PROGRAM STATE_MACHINE
VAR
	timer: TON;
END_VAR

IF ( CTRL.sdo = TRUE)THEN
	timer(IN:=TRUE);
	IF (timer.Q = TRUE) THEN
		CASE CTRL.in_opmode OF
			MODE.PROFILE_POSITION:
				Position_profile();	
			MODE.PROFILE_VELOCITY:
				Velocity_profile();
			MODE.TORQUE_PROFILE:
				Torque_profile();
			MODE.CYCLIC_SYNC_POS:
				Cyclic_sync_pos();
			MODE.CYCLIC_SYNC_VEL:
				Cyclic_sync_vel();
			MODE.CYCLIC_SYNC_TORQ:
				Cyclic_sync_torq();	
		ELSE
			CTRL.error:= PLC_ERROR.MODE_NO_SETUP;		
		END_CASE	
	END_IF
END_IF

END_PROGRAM

(* stored: Version 1.1.0.1, ProductVersion 3.1.4024.11
   POU STATE_MACHINE: Id {1a275fdd-adc3-4480-838a-4253a7626e42}, SpecialFunc None *)
